FUNCTION_BLOCK FB_MotionShareData IMPLEMENTS I_MotionShareData
VAR_INPUT
END_VAR
VAR_OUTPUT
END_VAR
VAR
END_VAR

{warning 'Add property implementation'}
PROPERTY AxisState : MC_AxisStates
GET
END_GET
END_PROPERTY

{warning 'Add property implementation'}
PROPERTY DriveEnable : BOOL
GET
END_GET
SET
END_SET
END_PROPERTY

{warning 'Add property implementation'}
PROPERTY ExecHome : BOOL
GET
END_GET
SET
END_SET
END_PROPERTY

{warning 'Add property implementation'}
PROPERTY ExecMove : BOOL
GET
END_GET
SET
END_SET
END_PROPERTY

{warning 'Add property implementation'}
PROPERTY GlobalReset : BOOL
GET
END_GET
SET
END_SET
END_PROPERTY

{warning 'Add property implementation'}
PROPERTY HomeBusy : BOOL
GET
END_GET
SET
END_SET
END_PROPERTY

{warning 'Add property implementation'}
PROPERTY LimBackward : BOOL
GET
END_GET
SET
END_SET
END_PROPERTY

{warning 'Add property implementation'}
PROPERTY LimForward : BOOL
GET
END_GET
SET
END_SET
END_PROPERTY

{warning 'Add property implementation'}
PROPERTY LimHit : BOOL
GET
END_GET
END_PROPERTY

{warning 'Add property implementation'}
PROPERTY LimHome : BOOL
GET
END_GET
SET
END_SET
END_PROPERTY

{warning 'Add property implementation'}
PROPERTY MoveBusy : BOOL
GET
END_GET
SET
END_SET
END_PROPERTY

{warning 'Add property implementation'}
PROPERTY NegativeDirection : BOOL
GET
END_GET
SET
END_SET
END_PROPERTY

{warning 'Add property implementation'}
PROPERTY NewMoveReq : BOOL
GET
END_GET
SET
END_SET
END_PROPERTY

{warning 'Add property implementation'}
PROPERTY PositiveDirection : BOOL
GET
END_GET
SET
END_SET
END_PROPERTY

{warning 'Add property implementation'}
PROPERTY ResetDone : BOOL
GET
END_GET
SET
END_SET
END_PROPERTY

{warning 'Add property implementation'}
PROPERTY RestoreDone : BOOL
GET
END_GET
SET
END_SET
END_PROPERTY

{warning 'Add property implementation'}
PROPERTY SavedPosition : LREAL
GET
END_GET
SET
END_SET
END_PROPERTY

{warning 'Add property implementation'}
PROPERTY ServoMode : BOOL
SET
END_SET
END_PROPERTY

END_FUNCTION_BLOCK

(* stored: Version 1.1.0.1
   POU FB_MotionShareData: Id {f8b65c5c-b9a7-4590-91d6-adb4de6e3c7e}, SpecialFunc None
   Property AxisState: Id {d176f804-fc0e-44b9-8e60-10d2b87b0348}
   Get Get: Id {75330f1e-001f-4b32-afc7-a6b00d9a0a05}
   Property DriveEnable: Id {dd065775-d061-4674-857b-1a465207cf2a}
   Get Get: Id {aae3f481-261b-4062-897f-695b55b2f21d}
   Set Set: Id {fc0de660-6e25-4bd5-9b11-4edda313922b}
   Property ExecHome: Id {8b17ab62-077b-43af-82ec-fac66a1f47f8}
   Get Get: Id {068a1a4e-8f6c-40ee-98a0-adc665c4ffb4}
   Set Set: Id {71528b05-c8de-4033-affd-66dda6137f8e}
   Property ExecMove: Id {afe566d9-cfc6-4b83-a641-12bf2b581a73}
   Get Get: Id {41ec7eba-dcf4-4649-87d9-d5dda5627497}
   Set Set: Id {138f7a45-745b-4a75-8201-7714b59a8ea5}
   Property GlobalReset: Id {95fc951b-8c55-425b-9a24-6e308eec1da7}
   Get Get: Id {771309ca-5d91-445c-877f-8024b89317ab}
   Set Set: Id {a9f8cb37-4851-4903-8e78-06c309a661a5}
   Property HomeBusy: Id {c8103306-69f6-440a-8cb9-173a6abd1584}
   Get Get: Id {13ad0c20-2d52-4a1e-8763-50106f6b8a65}
   Set Set: Id {fd61ff19-af24-4dfd-8140-67cda46e41a2}
   Property LimBackward: Id {20c5842a-0579-4ba4-a851-d8a4ee24523d}
   Get Get: Id {19d17128-ba41-4098-ae2f-878e456d188a}
   Set Set: Id {9298a045-01a1-4317-bf90-789d73d7a6f3}
   Property LimForward: Id {7a1f7e56-8919-4d10-8498-d2256e78a7ab}
   Get Get: Id {d4b57db0-bc7b-4f18-ac13-cf29af9c6233}
   Set Set: Id {2ead52aa-6c7c-42d5-aa5a-12f292bd7ad8}
   Property LimHit: Id {444df255-cede-4102-8dae-754c8f7ec8e0}
   Get Get: Id {2b291fce-ed83-49c3-98e9-64704f1192da}
   Property LimHome: Id {6cc35d0b-02a2-4059-83b5-53b0116285f1}
   Get Get: Id {f31c6006-ebec-4c16-ae71-1bbea4d60bc8}
   Set Set: Id {2c09ddde-1303-4d6b-a40b-8cd4fe86b5b4}
   Property MoveBusy: Id {e2a480ab-8340-4769-b50c-f6517912db82}
   Get Get: Id {15cdc1ab-d87a-4472-8a9d-50782f46bc57}
   Set Set: Id {aaaf2408-d259-4039-9124-203606d91335}
   Property NegativeDirection: Id {15d39468-6c3e-496a-8b79-93deae8d451f}
   Get Get: Id {2cc9ff11-6e17-412b-963b-a57070f6458a}
   Set Set: Id {a2af2ef5-89e8-4263-afe8-b89a52508fc8}
   Property NewMoveReq: Id {51dc54f4-66d7-4b9c-806d-30cd5ef37e4c}
   Get Get: Id {413954bd-54d7-4d6f-9572-222cb9276c2d}
   Set Set: Id {7e67fb6a-1267-436a-a823-62d30ef0003e}
   Property PositiveDirection: Id {bcfc651c-d34e-4ae0-9915-16e94869a276}
   Get Get: Id {998d7cff-5053-47a7-8095-db95a7b4b98a}
   Set Set: Id {1ff400a2-84e1-409e-b4be-23f2e232d3d6}
   Property ResetDone: Id {176381e7-6ff5-4d3e-9850-4d0383cbc218}
   Get Get: Id {d141e32b-2750-4f17-a33c-38458da09676}
   Set Set: Id {81df5bd6-9ef8-44f5-b2c7-6467b6f8d472}
   Property RestoreDone: Id {7b9b6bf3-2250-4f8c-ac2b-2577ae3a5f0d}
   Get Get: Id {6272c748-34d1-4e7f-b982-47dbc4329e14}
   Set Set: Id {30666cbe-8ea6-4027-ab37-ae59a9f109c6}
   Property SavedPosition: Id {85d18d09-48d0-431f-a598-c731c4ea0a10}
   Get Get: Id {573697f2-3242-496f-95b1-717a7b7505ac}
   Set Set: Id {647928d1-aa22-4fa1-a33f-67eeea507d40}
   Property ServoMode: Id {da8a21a2-5011-4334-90b7-7b4314c31378}
   Set Set: Id {552549cc-7fe0-4d06-b234-4039032415fd} *)
